Staubli VAL3: onF3Event.pgx

program onF3Event()
begin
  // look if the bButton is enable
  if bButton[2]
    // make the calibration


    ////    io:calibrate=true
    ////    delay(0.5)
    ////    io:calibrate=false


    //

    aioSet(MbAO_bResetErr,1)
    aioSet(MbAO_b8Axis,1)
    delay(0.5)
    aioSet(MbAO_b8Axis,0)
     call use:timerDialog("8轴已经复位",1)
    logMsg("[VALlaser] INTERFACE:7Axis Reset")
  endIf
end
